FUNCTION Convert_UINT_TO_DINT : Hresult
VAR_INPUT
	in : UINT;
	out : REFERENCE TO DINT;
END_VAR
VAR
	converted : DINT;
END_VAR
VAR CONSTANT
	INCOMPATIBLE : HRESULT := 16#9811070E;
END_VAR

converted := UINT_TO_DINT(in);

IF (DINT_TO_UINT(converted) <> in) THEN
	Convert_UINT_TO_DINT := INCOMPATIBLE;
	RETURN;
END_IF

out := converted;

END_FUNCTION

(* stored: Version 1.1.0.1, ProductVersion 3.1.4024.12
   POU Convert_UINT_TO_DINT: Id {323255d9-13c5-4457-9d25-977b03a40773}, SpecialFunc None *)
